(*********************************** G.D S.p.A. - Technical Department ***********************************
============= PROGRAM INFO ============
FOLDER:             TBD
MACHINES INVOLVED:  TBD 

============= DESCRIPTION =============
csp machine declaration

============= REVISIONS ===============
Date		Version	 	Author      	Description             
----------	-------		------------  	--------------------------------------------
2019/04/05 	0000.00	 	M.Grasso		Creation of the PRG

**********************************************************************************************************)
(*$R process_ref := prc; $*)
PROGRAM csp_case_feed_magazine_ls
VAR
	
	prc:											process;
	prc_path:										STRING;
	
END_VAR

_read_var_input();

_object_manager();

IF NOT objects_running()
THEN
	RETURN;	
END_IF

_read_process_image();

_mode_manager();

_set_runtime_properties();

(********************************* BODY *********************************)
(************************************************************************)

_handle_messages();

_write_output();

ACTION _handle_messages:
;
END_ACTION

ACTION _handle_process_test:
;
END_ACTION

ACTION _mode_manager:
IF process_mode_req_is_pending(prc)
THEN
    process_apply_mode_req_first_step(prc);
    CASE process_get_mode(prc) OF
        MODE_TO_ABSENT:
			;
        MODE_TO_INACTIVE:
			;
        MODE_TO_TEST:
			;
        MODE_TO_OPERATIONAL:
			;
    END_CASE
    process_apply_mode_req_second_step(prc);
END_IF
END_ACTION

ACTION _object_manager:
IF objects_initialization()
THEN
	sub_process_init(
		object_name					:= 'csp_case_feed_magazine_ls.prc', 
		process						:= csp_case_feed_magazine.prc, 
		CONVERSION_this				:= prc);
		
	prc_path 						:= process_get_path(prc);
END_IF

IF objects_running()
THEN
	process_cycle(prc);
END_IF
END_ACTION

ACTION _read_process_image:
;
END_ACTION

ACTION _read_var_input:
;
END_ACTION

ACTION _set_runtime_properties:
;
END_ACTION

ACTION _write_output:
;
END_ACTION

END_PROGRAM

(* stored: Version 1.1.0.1, ProductVersion 3.1.4022.12
   POU csp_case_feed_magazine_ls: Id {3f64a935-46b8-4c3c-a963-078544755c5f}, SpecialFunc None
   Action _handle_messages: Id {04433144-4736-4ad7-9d9f-a0125bd6fff1}
   Action _handle_process_test: Id {cac571f1-2ab2-421a-98e8-e52b62f46afe}
   Action _mode_manager: Id {011fbeca-0706-42ec-b695-d1e90d943079}
   Action _object_manager: Id {4bd8865f-1715-49ad-86e7-27210af5c081}
   Action _read_process_image: Id {18e4396c-233d-4364-97a6-054980508ffe}
   Action _read_var_input: Id {0c476b4a-a1af-4e54-92a1-f684ebd5e231}
   Action _set_runtime_properties: Id {471a9322-2729-401e-9102-22fc84cd7c3b}
   Action _write_output: Id {f83aec15-e5e8-40d3-9028-9f2eddf31286} *)
